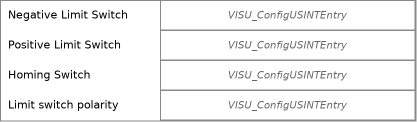
VISUALIZATION VISU_FaulhaberDriveConfig_LimitSwitches  // 417x122
VAR_IN_OUT
	active : FaulhaberDriveConfig;
	editable : FaulhaberDriveConfig;
END_VAR
    Label (5,0 135x30), "Negative Limit Switch"
    Frame (160,0 255x30)
        shows VISU_ConfigUSINTEntry(active := active.negativeLimitSwitch, editable := editable.negativeLimitSwitch)
    Label (5,30 135x30), "Positive Limit Switch"
    Frame (160,30 255x30)
        shows VISU_ConfigUSINTEntry(active := active.positiveLimitSwitch, editable := editable.positiveLimitSwitch)
    Label (5,60 135x30), "Homing Switch"
    Frame (160,60 255x30)
        shows VISU_ConfigUSINTEntry(active := active.homingSwitch, editable := editable.homingSwitch)
    Frame (160,90 255x30)
        shows VISU_ConfigUSINTEntry(active := active.limitSwitchPolarity, editable := editable.limitSwitchPolarity)
    Label (5,90 155x30), "Limit switch polarity"
END_VISUALIZATION

(* stored: Version 1.1.0.1, ProductVersion 3.1.4019.2
   Visu VISU_FaulhaberDriveConfig_LimitSwitches: Id {d0769472-1c77-4a4e-a904-4f2109bcd2bf} *)
